KUKA KRL program: RobotWarmup.src, RobotWarmup.dat

--- RobotWarmup.src ---
&ACCESS RVO
&REL 32
&PARAM EDITMASK = *
&PARAM TEMPLATE = C:\KRC\Roboter\Template\vorgabe
&PARAM DISKPATH = KRC:\R1
DEF RobotWarmup( )
DECL INT _nAns
;FOLD INI;%{PE}
  ;FOLD BASISTECH INI
    GLOBAL INTERRUPT DECL 3 WHEN $STOPMESS==TRUE DO IR_STOPM ( )
    INTERRUPT ON 3
    BAS (#INITMOV,0 )
  ;ENDFOLD (BASISTECH INI)
  ;FOLD USER INI
    ;Make your modifications here
    _nAns = 0

  ;ENDFOLD (USER INI)
  ;ENDFOLD (INI)

;************************************************
;              CNC Robotics Ltd
;              www.cncrobotics.co.uk
;************************************************
;     Contact: helpdesk@cncrobotics.co.uk
;     Date: 05/04/24
;     Version: 0.21.54
;************************************************
; Description: Routine to warm up the robot
;************************************************

; Warning message to the user before warmup starts
MsgDialog(_nAns,"Ensure the robot is in a clear area and wont crash during warm-up.","Robot",,,,,,,"Exit","Continue", FALSE, nRobotMsg + 6, E_progCommonMsgOpt)

IF (_nAns == 1) THEN
   _nAns = 0
ELSE
	RETURN
ENDIF

;Loop until A1 motor is above 314 degrees kelvin
LOOP

;Move to home
;FOLD PTP HOME CONT Vel=100 % DEFAULT ;%{PE}
;FOLD Parameters ;%{h}
;Params IlfProvider=kukaroboter.basistech.inlineforms.movement.old; Kuka.IsGlobalPoint=False; Kuka.PointName=HOME; Kuka.BlendingEnabled=True; Kuka.MoveDataPtpName=DEFAULT; Kuka.VelocityPtp=100; Kuka.CurrentCDSetIndex=0; Kuka.MovementParameterFieldEnabled=True; IlfCommand=PTP
;ENDFOLD
$BWDSTART = FALSE
PDAT_ACT = PDEFAULT
FDAT_ACT = FHOME
BAS(#PTP_PARAMS, 100.0)
SET_CD_PARAMS (0)
PTP XHOME C_Dis
;ENDFOLD

;Move to other position of warmup
;FOLD PTP P1 CONT Vel=100 % PDAT1 Tool[0] Base[0] ;%{PE}
;FOLD Parameters ;%{h}
;Params IlfProvider=kukaroboter.basistech.inlineforms.movement.old; Kuka.IsGlobalPoint=False; Kuka.PointName=P1; Kuka.BlendingEnabled=True; Kuka.MoveDataPtpName=PDAT1; Kuka.VelocityPtp=100; Kuka.CurrentCDSetIndex=0; Kuka.MovementParameterFieldEnabled=True; IlfCommand=PTP
;ENDFOLD
$BWDSTART = FALSE
PDAT_ACT = PPDAT1
FDAT_ACT = FP1
BAS(#PTP_PARAMS, 100.0)
SET_CD_PARAMS (0)
PTP XP1 C_Dis
;ENDFOLD

	;When A1 motor temp reaches 314 degrees, end warmup and move home
	IF ($MOT_TEMP[1] >314) THEN
		MsgNotify("Robot warmup complete.", "Robot",,, nRobotMsg + 7, E_progNotifyMsgOpt)
		HomePosition()
		RETURN
	ENDIF

ENDLOOP

END

--- RobotWarmup.dat ---
&ACCESS  RVP
&PARAM EDITMASK = *
&PARAM TEMPLATE = C:\KRC\Roboter\Template\vorgabe
&PARAM DISKPATH = KRC:\R1
&REL 29
DEFDAT  ROBOTWARMUP
;FOLD EXTERNAL DECLARATIONS;%{PE}%MKUKATPBASIS,%CEXT,%VCOMMON,%P
;FOLD BASISTECH EXT;%{PE}%MKUKATPBASIS,%CEXT,%VEXT,%P
EXT  BAS (BAS_COMMAND  :IN,REAL  :IN )
DECL INT SUCCESS
;ENDFOLD (BASISTECH EXT)
;FOLD USER EXT;%{E}%MKUKATPUSER,%CEXT,%VEXT,%P
;Make your modifications here

;ENDFOLD (USER EXT)
;ENDFOLD (EXTERNAL DECLARATIONS)
DECL E6POS XP1={X 1538.34753,Y -747.365540,Z 1379.56494,A 177.447876,B 89.2426224,C 177.449707,S 22,T 50,E1 0.627261639,E2 0.0,E3 0.0,E4 0.0,E5 0.0,E6 0.0}
DECL FDAT FP1={TOOL_NO 0,BASE_NO 0,IPO_FRAME #BASE,POINT2[] " "}
DECL PDAT PPDAT1={VEL 100.000,ACC 100.000,APO_DIST 500.000,APO_MODE #CDIS,GEAR_JERK 100.000,EXAX_IGN 0}
DECL MODULEPARAM_T LAST_TP_PARAMS={PARAMS[] "Kuka.PointName=P1; Kuka.FrameData.base_no=0; Kuka.FrameData.tool_no=0; Kuka.FrameData.ipo_frame=#BASE; Kuka.isglobalpoint=False; Kuka.MoveDataPtpName=PDAT1; Kuka.MovementDataPdat.apo_mode=#CDIS; Kuka.MovementDataPdat.apo_dist=500; Kuka.MovementData.vel=100; Kuka.MovementData.acc=100; Kuka.MovementData.exax_ign=0; Kuka.VelocityPtp=100; Kuka.BlendingEnabled=True; Kuka.CurrentCDSetIndex=0; Kuka.FrameData.point2=; Kuka.VelocityFieldEnabled=True; Kuka.ColDetectFieldEnabled=False; Kuka.MovementParameterFieldEnabled=True; Kuka.IsAngleEnabled=False; Kuka.APXEnabled=False"}
ENDDAT
